   // Stellrückmeldungen
   "UP_CM03.GP03".In.SRM_Saugseite_auf := "E_SRM_CM03.QM33_auf" AND NOT "E_SRM_CM03.QM33_zu";
   "UP_CM03.GP03".In.SRM_Saugseite_zu := "E_SRM_CM03.QM33_zu" AND NOT "E_SRM_CM03.QM33_auf";
   "UP_CM03.GP03".In.SRM_Druckseite_auf := "E_SRM_CM03.QM34_auf" AND NOT "E_SRM_CM03.QM34_zu";
   "UP_CM03.GP03".In.SRM_Druckseite_zu := "E_SRM_CM03.QM34_zu" AND NOT "E_SRM_CM03.QM34_auf";

   "UP_CM03.GP03".In.GW_p_UP := "E_GW_p_CM03.BP05";
   // TW senkt
   "UP_CM03.GP03".In.TW_senkt := ("DB_POS".POS[7].FW_Senkt OR "DB_POS".POS[8].FW_Senkt OR "DB_POS".POS[9].FW_Senkt
   OR "DB_POS".POS[10].FW_Senkt OR "DB_POS".POS[11].FW_Senkt OR "DB_POS".POS[12].FW_Senkt) AND "DI_FW_1".ZST.Mittig;

   // Frequenzumrichter [Index 3]
   "UP_CM03.GP03".In.FU_speed := "FU_In_Out".FU[3].PE.Speed;
   "UP_CM03.GP03".In.FU_betriebsbereit := "FU_In_Out".FU[3].PE.Statusbyte.Bereit;
   "UP_CM03.GP03".In.FU_Stoerung := "FU_In_Out".FU[3].PE.Statusbyte.Stoer;
   "UP_CM03.GP03".Param.SW_Hand := "Panel".UP_CM03.SW_Hand;
   "UP_CM03.GP03".Param.SW_Auto_AZ := "Panel".UP_CM03.SW_Auto_AZ;
   "UP_CM03.GP03".Param.SW_Auto_aAZ := "Panel".UP_CM03.SW_Auto_aAZ;

   // Hand
   "UP_CM03.GP03".In.Ein := "Panel".UP_CM03.Ein;
   // Auto
   "UP_CM03.GP03".In.Auto := FALSE; // "Panel".UP_CM03.Auto;
   // Betriebsart
   "UP_CM03.GP03".In.Betriebsart := "Panel".UP_CM03.BA;
   // Spülzeit
   "UP_CM03.GP03".Param.Spülzeit := DINT_TO_TIME(INT_TO_DINT("Panel".UP_CM03.Sp_Ventil.Sollzeit) * 1000);
   // Drucktest
   "UP_CM03.GP03".Param.DT_Druckaufbau := T#1m;
   "UP_CM03.GP03".Param.SW_Drucktest := "Panel".UP_CM03.Drucktest.Solldruck;
   "UP_CM03.GP03".Param.DT_Testzeit := DINT_TO_TIME(INT_TO_DINT("Panel".UP_CM03.Drucktest.Sollzeit) * 1000);


   // --> Panel
   "Panel".CM03.Niv_TGS := "UP_CM03.GP03".In.Niv_TLS;
   "Panel".CM03.Niv_Min := "UP_CM03.GP03".In.Niv_min;
   "Panel".CM03.GW_p_UP := "UP_CM03.GP03".In.GW_p_UP;
   "Panel".CM03.Niv_Proz := "UP_CM03.GP03".Zst.Niveau;
   "Panel".UP_CM03.Sp_Ventil.Restzeit := TIME_TO_INT("UP_CM03.GP03".Zst.Restzeit_Spülen / 1000);
   "Panel".UP_CM03.Drucktest.Restzeit := TIME_TO_INT("UP_CM03.GP03".Zst.Restzeit_DT / 1000);
   "Panel".UP_CM03.Drucktest.Schritt := "UP_CM03.GP03".Zst.Status_DT;
   "Panel".UP_CM03.Status := "UP_CM03.GP03".Zst.Status_GP0x;
   "Panel".UP_CM03.speed := "UP_CM03.GP03".Zst.speed;
   "Panel".UP_CM03.Bedienung_Erlaubt := "UP_CM03.GP03".Zst.Bedienung_erlaubt;
END_REGION

REGION Network 6 (SCL): CM04
   "UP_CM04.GP06".Param.Name := 'UP_CM04.GP06';
   // Niveaus
   "UP_CM04.GP06".In.Niv_TLS := "E_Niv_TLS_CM04.BL14";
   "UP_CM04.GP06".In.Niv_min := "E_Niv_Min_CM04.BL13";
   "UP_CM04.GP06".In.Frg_Niv_CM05 := NOT "Pu_CM05.GP11_DB".In."Niv_max_CM05.BL01" AND NOT "Pu_CM05.GP11_DB".In."Niv_Uel_CM05.BL05";
   "UP_CM04.GP06".In.ext_Freigabe := "E_Al_Gas_ok" AND NOT "E_Not-Strom";
   // Ist-Druck
   "UP_CM04.GP06".In.Druck_Pumpe := "Panel".IW."p_CM04.BP08";

   // Stellrückmeldungen
   "UP_CM04.GP06".In.SRM_Saugseite_auf := "E_SRM_CM04.QM72_auf" AND NOT "E_SRM_CM04.QM72_zu";
   "UP_CM04.GP06".In.SRM_Saugseite_zu := "E_SRM_CM04.QM72_zu" AND NOT "E_SRM_CM04.QM72_auf";
   "UP_CM04.GP06".In.SRM_Druckseite_auf := "E_SRM_CM04.QM73_auf" AND NOT "E_SRM_CM04.QM73_zu";
   "UP_CM04.GP06".In.SRM_Druckseite_zu := "E_SRM_CM04.QM73_zu" AND NOT "E_SRM_CM04.QM73_auf";

   "UP_CM04.GP06".In.GW_p_UP := "E_GW_p_CM04.BP08";

   // TW senkt
   "UP_CM04.GP06".In.TW_senkt := ("DB_POS".POS[19].FW_Senkt OR "DB_POS".POS[20].FW_Senkt OR "DB_POS".POS[21].FW_Senkt
   OR "DB_POS".POS[22].FW_Senkt OR "DB_POS".POS[23].FW_Senkt OR "DB_POS".POS[24].FW_Senkt) AND "DI_FW_1".ZST.Mittig;

   // Frequenzumrichter [Index 6]
   "UP_CM04.GP06".In.FU_speed := "FU_In_Out".FU[6].PE.Speed;
   "UP_CM04.GP06".In.FU_betriebsbereit := "FU_In_Out".FU[6].PE.Statusbyte.Bereit;
   "UP_CM04.GP06".In.FU_Stoerung := "FU_In_Out".FU[6].PE.Statusbyte.Stoer;
   "UP_CM04.GP06".Param.SW_Hand := "Panel".UP_CM04.SW_Hand;
   "UP_CM04.GP06".Param.SW_Auto_AZ := "Panel".UP_CM04.SW_Auto_AZ;
   "UP_CM04.GP06".Param.SW_Auto_aAZ := "Panel".UP_CM04.SW_Auto_aAZ;

   // Hand
   "UP_CM04.GP06".In.Ein := "Panel".UP_CM04.Ein;
   // Auto
   "UP_CM04.GP06".In.Auto := FALSE; // "Panel".UP_CM04.Auto;
   // Betriebsart
   "UP_CM04.GP06".In.Betriebsart := "Panel".UP_CM04.BA;

   // Spülzeit
   "UP_CM04.GP06".Param.Spülzeit := DINT_TO_TIME(INT_TO_DINT("Panel".UP_CM04.Sp_Ventil.Sollzeit) * 1000);
   // Drucktest
   "UP_CM04.GP06".Param.DT_Druckaufbau := T#1m;
   "UP_CM04.GP06".Param.SW_Drucktest := "Panel".UP_CM04.Drucktest.Solldruck;
   "UP_CM04.GP06".Param.DT_Testzeit := DINT_TO_TIME(INT_TO_DINT("Panel".UP_CM04.Drucktest.Sollzeit) * 1000);

   // --> Panel
   "Panel".CM04.Niv_TGS := "UP_CM04.GP06".In.Niv_TLS;
   "Panel".CM04.Niv_Min := "UP_CM04.GP06".In.Niv_min;
   "Panel".CM04.GW_p_UP := "UP_CM04.GP06".In.GW_p_UP;
   "Panel".CM04.Niv_Proz := "UP_CM04.GP06".Zst.Niveau;
   "Panel".UP_CM04.Sp_Ventil.Restzeit := TIME_TO_INT("UP_CM04.GP06".Zst.Restzeit_Spülen / 1000);
   "Panel".UP_CM04.Drucktest.Restzeit := TIME_TO_INT("UP_CM04.GP06".Zst.Restzeit_DT / 1000);
   "Panel".UP_CM04.Drucktest.Schritt := "UP_CM04.GP06".Zst.Status_DT;
   "Panel".UP_CM04.Status := "UP_CM04.GP06".Zst.Status_GP0x;
   "Panel".UP_CM04.speed := "UP_CM04.GP06".Zst.speed;
   "Panel".UP_CM04.Bedienung_Erlaubt := "UP_CM04.GP06".Zst.Bedienung_erlaubt;
END_REGION

REGION Network 7 (SCL): CM05
   // Motorschutzschalter
   "Pu_CM05.GP11_DB".In.MSS_ok := "E_MSS_ok_CM05.GP11";
   // Druckschalter
   "Pu_CM05.GP11_DB".In.GW_p := "E_GW_p_CM05.BP09";
   // Ist-Druck
   "Pu_CM05.GP11_DB".In.Druck_Pumpe :="Panel".IW."p_CM05.BP09";

   // Niveaus
   "Pu_CM05.GP11_DB".In."Niv_max_CM05.BL01" := "E_Niv_max_CM05.BL01";
   "Pu_CM05.GP11_DB".In."Niv_min_CM05.BL02" := "E_Niv_min_CM05.BL02";
   "Pu_CM05.GP11_DB".In."Niv_TLS_CM05.BL03" := "E_Niv_TLS_CM05.BL03";
   "Pu_CM05.GP11_DB".In."Niv_Uel_CM05.BL05" :=  NOT "E_Niv_Uel_CM05.BL12";

   // Stellrückmeldungen
   "Pu_CM05.GP11_DB".In."SRM_CM05.QM61_auf" := "E_SRM_CM05.QM61_auf" AND NOT "E_SRM_CM05.QM61_zu";
   "Pu_CM05.GP11_DB".In."SRM_CM05.QM61_zu" := "E_SRM_CM05.QM61_zu" AND NOT "E_SRM_CM05.QM61_auf";
   "Pu_CM05.GP11_DB".In."SRM_CM05.QM64_auf" := "E_SRM_CM05.QM64_auf" AND NOT "E_SRM_CM05.QM64_zu";
   "Pu_CM05.GP11_DB".In."SRM_CM05.QM64_zu" := "E_SRM_CM05.QM64_zu"  AND NOT "E_SRM_CM05.QM64_auf";

   // Neutra
   "Pu_CM05.GP11_DB".In.AWA_ok := "E_AWA_ok";
   "Pu_CM05.GP11_DB".In.Frg_AWA := "E_Frg_AWA";
   // Hand
   "Pu_CM05.GP11_DB".In.Ein := "Panel".Pu_CM05.Ein;
   // Auto
   "Pu_CM05.GP11_DB".In.Auto := "Panel".Pu_CM05.Auto;
   // Betriebsart
   "Pu_CM05.GP11_DB".In.Betriebsart := "Panel".Pu_CM05.BA;
   // Spülzeit
   "Pu_CM05.GP11_DB".Param.Spülzeit := DINT_TO_TIME(INT_TO_DINT("Panel".Pu_CM05.Sp_Ventil.Sollzeit) * 1000);
   // Drucktest
   "Pu_CM05.GP11_DB".Param.DT_Druckaufbau := T#1m;
   "Pu_CM05.GP11_DB".Param.SW_Drucktest := "Panel".Pu_CM05.Drucktest.Solldruck;
   "Pu_CM05.GP11_DB".Param.DT_Testzeit := DINT_TO_TIME(INT_TO_DINT("Panel".Pu_CM05.Drucktest.Sollzeit) * 1000);

   // --> Panel
   "Panel".CM05.GW_p_Pu := "Pu_CM05.GP11_DB".In.GW_p;
   "Panel".CM05.Niv_Proz := "Pu_CM05.GP11_DB".Zst.Niveau;
   "Panel".CM05.Niv_TGS := "Pu_CM05.GP11_DB".In."Niv_TLS_CM05.BL03";
   "Panel".CM05.Niv_Min := "Pu_CM05.GP11_DB".In."Niv_min_CM05.BL02";
   "Panel".CM05.Niv_max := "Pu_CM05.GP11_DB".In."Niv_max_CM05.BL01";
   "Panel".CM05.Niv_Uel := "Pu_CM05.GP11_DB".In."Niv_Uel_CM05.BL05";
   "Panel".Pu_CM05.Sp_Ventil.Restzeit := TIME_TO_INT("Pu_CM05.GP11_DB".Zst.Restzeit_Spülen / 1000);
   "Panel".Pu_CM05.Drucktest.Restzeit := TIME_TO_INT("Pu_CM05.GP11_DB".Zst.Restzeit_DT / 1000);
   "Panel".Pu_CM05.Drucktest.Schritt := "Pu_CM05.GP11_DB".Zst.Status_DT;
   "Panel".Pu_CM05.Status := "Pu_CM05.GP11_DB".Zst.Status_GP11;
   "Panel".CM05.AWA_Bereit := "Pu_CM05.GP11_DB".In.AWA_ok;
   "Panel".CM05.Frg_Abpumpen := "Pu_CM05.GP11_DB".In.Frg_AWA;
   "Panel".Pu_CM05.Bedienung_Erlaubt := "Pu_CM05.GP11_DB".Zst.Bedienung_erlaubt;
END_REGION

REGION Network 8 (SCL): CL0x
   //CL01
   // Niveaus
   "Pu_CL01.GP08".In.Frg_Niv_CM05 :=  NOT "Pu_CM05.GP11_DB".In."Niv_max_CM05.BL01" AND NOT "Pu_CM05.GP11_DB".In."Niv_Uel_CM05.BL05";
   "Pu_CL01.GP08".In.Leckage_ok := "E_LS_CL01.BL28";
   // Hand
   "Pu_CL01.GP08".In.Ein :="Panel".Pu_CL01.Ein;
   // Auto
   "Pu_CL01.GP08".In.Auto := "Panel".Pu_CL01.Auto;
   // Betriebsart
   "Pu_CL01.GP08".In.Betriebsart := "Panel".Pu_CL01.BA;
   // Spülzeit
   "Pu_CL01.GP08".Param.Spülzeit := DINT_TO_TIME(INT_TO_DINT("Panel".Pu_CL01.Sp_Ventil.Sollzeit) * 1000);

   // --> Panel
   "Panel".CL0x."LS_CL01.BL28" := NOT "Pu_CL01.GP08".In.Leckage_ok;
   "Panel".CL0x.Niv_Proz_CL01 := "Pu_CL01.GP08".Zst.Niveau;
   "Panel".Pu_CL01.Sp_Ventil.Restzeit := TIME_TO_INT("Pu_CL01.GP08".Zst.Restzeit_Spülen / 1000);
   "Panel".Pu_CL01.Status := "Pu_CL01.GP08".Zst.Status_GP0x;
   "Panel".Pu_CL01.Bedienung_Erlaubt := "Pu_CL01.GP08".Zst.Bedienung_Erlaubt;

   //CL02
   // Niveaus
   "Pu_CL02.GP09".In.Frg_Niv_CM05 :=  NOT "Pu_CM05.GP11_DB".In."Niv_max_CM05.BL01" AND NOT "Pu_CM05.GP11_DB".In."Niv_Uel_CM05.BL05";
   "Pu_CL02.GP09".In.Leckage_ok := "E_LS_CL02.BL29";
   // Hand
   "Pu_CL02.GP09".In.Ein := "Panel".Pu_CL02.Ein;
   // Auto
   "Pu_CL02.GP09".In.Auto := "Panel".Pu_CL02.Auto;
   // Betriebsart
   "Pu_CL02.GP09".In.Betriebsart := "Panel".Pu_CL02.BA;
   // Spülzeit
   "Pu_CL02.GP09".Param.Spülzeit := DINT_TO_TIME(INT_TO_DINT("Panel".Pu_CL02.Sp_Ventil.Sollzeit) * 1000);

   // --> Panel
   "Panel".CL0x."LS_CL02.BL29" := NOT  "Pu_CL02.GP09".In.Leckage_ok;
   "Panel".CL0x.Niv_Proz_CL02 := "Pu_CL02.GP09".Zst.Niveau;
   "Panel".Pu_CL02.Sp_Ventil.Restzeit := TIME_TO_INT("Pu_CL02.GP09".Zst.Restzeit_Spülen / 1000);
   "Panel".Pu_CL02.Status := "Pu_CL02.GP09".Zst.Status_GP0x;
   "Panel".Pu_CL02.Bedienung_Erlaubt := "Pu_CL02.GP09".Zst.Bedienung_Erlaubt;
END_REGION

REGION Network 9 (SCL): GP01
   // Versorgung
   //Niveaus
   "Pu_GP01.GP13".In.Niv_min := "E_Niv_min_GP01.BL17";
   "Pu_GP01.GP13".In.Niv_max := NOT "E_Niv_max_GP01.BL20";
   "Pu_GP01.GP13".In.Niveau := INT_TO_USINT(REAL_TO_INT("Panel".IW."Niv_GP01.BL30"));
   // Leckagesensoren
   "Pu_GP01.GP13".In.Leckage_Pumpe_ok := NOT "E_LS_GP01.BL15";
   "Pu_GP01.GP13".In.Leckage_PFA_Uebergang_ok := "E_LS_GP01.BL16";
   "Pu_GP01.GP13".In.Leckage_Doppelrohr_ok := "E_LS_GP01.BL19";
   "Pu_GP01.GP13".In.Leckage_Uml_Tunnel_ok := "E_LS_GP01.BL34";
   "Pu_GP01.GP13".In.Leckage_Doppelschlauch_ok := TRUE; // nur GP02
   "Pu_GP01.GP13".In.kein_Gas_Alarm := "E_Al_Gas_ok";

   "Pu_GP01.GP13".In.Niv_Min_CM01 := "E_Niv_Min_CM01.BL03";
   "Pu_GP01.GP13".In.Niv_Max_CM01 := "E_Niv_Max_CM01.BL02";
   "Pu_GP01.GP13".In.Niv_Übervoll_CM01 := NOT "E_Niv_UeL_CM01.BL01";
   "Pu_GP01.GP13".In.Niv_Min_CM02 := "E_Niv_Min_CM02.BL10";
   "Pu_GP01.GP13".In.Niv_Max_CM02 := "E_Niv_Max_CM02.BL09";
   "Pu_GP01.GP13".In.Niv_Übervoll_CM02 := NOT "E_Niv_UeL_CM02.BL08";
   "Pu_GP01.GP13".In.Frg_Niv_CM05 := NOT "Pu_CM05.GP11_DB".In."Niv_max_CM05.BL01" AND NOT "Pu_CM05.GP11_DB".In."Niv_Uel_CM05.BL05";

   // Stellrückmeldungen
   "Pu_GP01.GP13".In.SRM_Saugseite_auf := "E_SRM_GP01.QM15_auf" AND NOT "E_SRM_GP01.QM15_zu";
   "Pu_GP01.GP13".In.SRM_Saugseite_zu := "E_SRM_GP01.QM15_zu" AND NOT "E_SRM_GP01.QM15_auf";
   "Pu_GP01.GP13".In.SRM_Druckseite_auf := "E_SRM_GP01.QM18_auf" AND NOT "E_SRM_GP01.QM18_zu";
   "Pu_GP01.GP13".In.SRM_Druckseite_zu := "E_SRM_GP01.QM18_zu" AND NOT "E_SRM_GP01.QM18_auf";
   "Pu_GP01.GP13".In.SRM_Eingang_Spülltg_auf := "E_SRM_GP01.QM16_auf" AND NOT "E_SRM_GP01.QM16_zu";
   "Pu_GP01.GP13".In.SRM_Eingang_Spülltg_zu := "E_SRM_GP01.QM16_zu" AND NOT "E_SRM_GP01.QM16_auf";
   "Pu_GP01.GP13".In.SRM_Ausgang_Spülltg_auf := "E_SRM_GP01.QM17_auf" AND NOT "E_SRM_GP01.QM17_zu";
   "Pu_GP01.GP13".In.SRM_Ausgang_Spülltg_zu := "E_SRM_GP01.QM17_zu" AND NOT "E_SRM_GP01.QM17_auf";
   "Pu_GP01.GP13".In.SRM_Versogung_UV01_auf := "E_SRM_GP01.QM22_auf" AND NOT "E_SRM_GP01.QM22_zu";
   "Pu_GP01.GP13".In.SRM_Versogung_UV01_zu := "E_SRM_GP01.QM22_zu" AND NOT "E_SRM_GP01.QM22_auf";
   "Pu_GP01.GP13".In.SRM_UV01_CM01_auf := "E_SRM_GP01.QM20_auf" AND NOT "E_SRM_GP01.QM20_zu";
   "Pu_GP01.GP13".In.SRM_UV01_CM01_zu := "E_SRM_GP01.QM20_zu" AND NOT "E_SRM_GP01.QM20_auf";
   "Pu_GP01.GP13".In.SRM_UV01_CM02_auf := "E_SRM_GP01.QM19_auf" AND NOT "E_SRM_GP01.QM19_zu";
   "Pu_GP01.GP13".In.SRM_UV01_CM02_zu := "E_SRM_GP01.QM19_zu" AND NOT "E_SRM_GP01.QM19_auf";

   "Pu_GP01.GP13".In.IBC_vorhanden := "E_S_IBC_GP01.BG21";
   "Pu_GP01.GP13".In.Tuer_vorn_zu := "DB_PNOZ_IN_Out".In.Tuer_zu_vorn_GP01;
   "Pu_GP01.GP13".In.Tuer_seitlich_zu := "DB_PNOZ_IN_Out".In.Tuer_zu_Seite_GP01;

   "Pu_GP01.GP13".In.GW_Dfl := "E_GW_Dfl_GP01.BF01";
   "Pu_GP01.GP13".In.Imp_Dfl := "E_Imp_GP01.BF01";
   "Pu_GP01.GP13".In.Quitt_Al_Dfl := "DB_ANLAGE".IN.Quitt_Err;
   "Pu_GP01.GP13".In.Dfl := "Panel".IW."Dfl_GP01.BF01";

   // Hand
   "Pu_GP01.GP13".In.Ein := "Panel".Pu_Vers_GP01.Ein;
   // Auto
   "Pu_GP01.GP13".In.Auto := "Panel".Pu_Vers_GP01.Auto;
   // Betriebsart
   "Pu_GP01.GP13".In.Betriebsart := "Panel".Pu_Vers_GP01.BA;
   // Spülzeit
   "Pu_GP01.GP13".Param.Spülzeit := DINT_TO_TIME(INT_TO_DINT("Panel".Pu_Vers_GP01.Sp_Ventil.Sollzeit) * 1000);

   // --> Panel
   "Panel".GP01.Niv_leer := "Pu_GP01.GP13".In.Niv_min;
   "Panel".GP01.Niv_max := "Pu_GP01.GP13".In.Niv_max;
   "Panel".GP01.IBC_vorhanden := "Pu_GP01.GP13".In.IBC_vorhanden;
   "Panel".GP01.Tür_zu_vorn := "Pu_GP01.GP13".In.Tuer_vorn_zu;
   "Panel".GP01.Tür_zu_seitlich := "Pu_GP01.GP13".In.Tuer_seitlich_zu;

   "Panel".GP01.LS_Pumpe := NOT "Pu_GP01.GP13".In.Leckage_Pumpe_ok;
   "Panel".GP01.LS_Doppelrohr_BL19 := NOT "Pu_GP01.GP13".In.Leckage_Doppelrohr_ok;
   "Panel".GP01.LS_PFA_Übergang := NOT "Pu_GP01.GP13".In.Leckage_PFA_Uebergang_ok;
   "Panel".GP01.LS_Uml_Tunnel := NOT "Pu_GP01.GP13".In.Leckage_Uml_Tunnel_ok;

   "Panel".GP01.Niv_Proz := "Pu_GP01.GP13".In.Niveau;

   "Panel".GP01.Versorgung := "Pu_GP01.GP13".In.Betriebsart < 4;
   "Panel".GP01.Entsorgung := "Pu_GP01.GP13".In.Betriebsart = 4;


   "Panel".Pu_Vers_GP01.Status := "Pu_GP01.GP13".Zst.Status_GP0x;
   "Panel".Pu_Vers_GP01.Sp_Ventil.Restzeit := TIME_TO_INT("Pu_GP01.GP13".Zst.Restzeit_Spülen / 1000);
   "Panel".Pu_Vers_GP01.Bedienung_Erlaubt := "Pu_GP01.GP13".Zst.Bedienung_erlaubt;
   //-----------------------------------------------------------------------------------------------------------------------------------------
   // Abpumpen
   // Niveaus
   "Pu_GP01.GP12".In.Frg_Niv_CM05 :=  NOT "Pu_CM05.GP11_DB".In."Niv_max_CM05.BL01" AND NOT "Pu_CM05.GP11_DB".In."Niv_Uel_CM05.BL05";
   "Pu_GP01.GP12".In.Leckage_ok := "E_LS_GP01.BL18";
   // Hand
   "Pu_GP01.GP12".In.Ein := "Panel".Pu_Entl_GP01.Ein;
   // Auto
   "Pu_GP01.GP12".In.Auto := "Panel".Pu_Entl_GP01.Auto;
   // Betriebsart
   "Pu_GP01.GP12".In.Betriebsart := "Panel".Pu_Entl_GP01.BA;
   // Spülzeit
   "Pu_GP01.GP12".Param.Spülzeit := DINT_TO_TIME(INT_TO_DINT("Panel".Pu_Entl_GP01.Sp_Ventil.Sollzeit) * 1000);

   // --> Panel
   "Panel".GP01.LS_PuSu := NOT "Pu_GP01.GP12".In.Leckage_ok;
   "Panel".Pu_Entl_GP01.Sp_Ventil.Restzeit := TIME_TO_INT("Pu_GP01.GP12".Zst.Restzeit_Spülen / 1000);
   "Panel".Pu_Entl_GP01.Status := "Pu_GP01.GP12".Zst.Status_GP0x;
   "Panel".Pu_Entl_GP01.Bedienung_Erlaubt := "Pu_GP01.GP12".Zst.Bedienung_Erlaubt;
END_REGION

REGION Network 10 (SCL): GP02
   // Versorgung
   //Niveaus
   "Pu_GP02.GP10".In.Niv_min := "E_Niv_min_GP02.BL24";
   "Pu_GP02.GP10".In.Niv_max := NOT "E_Niv_max_GP02.BL23";
   "Pu_GP02.GP10".In.Niveau := INT_TO_USINT(REAL_TO_INT("Panel".IW."Niv_GP02.BL31"));
   // Leckagesensoren
   "Pu_GP02.GP10".In.Leckage_Pumpe_ok := NOT "E_LS_GP02.BL27";
   "Pu_GP02.GP10".In.Leckage_PFA_Uebergang_ok := "E_LS_GP02.BL25";
   "Pu_GP02.GP10".In.Leckage_Doppelrohr_ok := "E_LS_GP01.BL19";
   "Pu_GP02.GP10".In.Leckage_Uml_Tunnel_ok := TRUE; // nur GP01
   "Pu_GP02.GP10".In.Leckage_Doppelschlauch_ok := "E_LS_GP02.BL32";
   "Pu_GP02.GP10".In.kein_Gas_Alarm := "E_Al_Gas_ok";

   "Pu_GP02.GP10".In.Niv_Min_CM01 := "E_Niv_Min_CM01.BL03";
   "Pu_GP02.GP10".In.Niv_Max_CM01 := "E_Niv_Max_CM01.BL02";
   "Pu_GP02.GP10".In.Niv_Übervoll_CM01 := NOT "E_Niv_UeL_CM01.BL01";
   "Pu_GP02.GP10".In.Niv_Min_CM02 := "E_Niv_Min_CM02.BL10";
   "Pu_GP02.GP10".In.Niv_Max_CM02 := "E_Niv_Max_CM02.BL09";
   "Pu_GP02.GP10".In.Niv_Übervoll_CM02 := NOT "E_Niv_UeL_CM02.BL08";
   "Pu_GP02.GP10".In.Frg_Niv_CM05 := NOT "Pu_CM05.GP11_DB".In."Niv_max_CM05.BL01" AND NOT "Pu_CM05.GP11_DB".In."Niv_Uel_CM05.BL05";

   // Stellrückmeldungen
   "Pu_GP02.GP10".In.SRM_Saugseite_auf := "E_SRM_GP02.QM38_auf" AND NOT "E_SRM_GP02.QM38_zu";
   "Pu_GP02.GP10".In.SRM_Saugseite_zu := "E_SRM_GP02.QM38_zu" AND NOT "E_SRM_GP02.QM38_auf";
   "Pu_GP02.GP10".In.SRM_Druckseite_auf := "E_SRM_GP02.QM40_auf" AND NOT "E_SRM_GP02.QM40_zu";
   "Pu_GP02.GP10".In.SRM_Druckseite_zu := "E_SRM_GP02.QM40_zu" AND NOT "E_SRM_GP02.QM40_auf";
   "Pu_GP02.GP10".In.SRM_Eingang_Spülltg_auf := "E_SRM_GP02.QM39_auf" AND NOT "E_SRM_GP02.QM39_zu";
   "Pu_GP02.GP10".In.SRM_Eingang_Spülltg_zu := "E_SRM_GP02.QM39_zu" AND NOT "E_SRM_GP02.QM39_auf";
   "Pu_GP02.GP10".In.SRM_Ausgang_Spülltg_auf := "E_SRM_GP02.QM42_auf" AND NOT "E_SRM_GP02.QM42_zu";
   "Pu_GP02.GP10".In.SRM_Ausgang_Spülltg_zu := "E_SRM_GP02.QM42_zu" AND NOT "E_SRM_GP02.QM42_auf";
   "Pu_GP02.GP10".In.SRM_Versogung_UV01_auf := "E_SRM_GP01.QM21_auf" AND NOT "E_SRM_GP01.QM21_zu";
   "Pu_GP02.GP10".In.SRM_Versogung_UV01_zu := "E_SRM_GP01.QM21_zu" AND NOT "E_SRM_GP01.QM21_auf";
   "Pu_GP02.GP10".In.SRM_UV01_CM01_auf := "E_SRM_GP01.QM20_auf" AND NOT "E_SRM_GP01.QM20_zu";
   "Pu_GP02.GP10".In.SRM_UV01_CM01_zu := "E_SRM_GP01.QM20_zu" AND NOT "E_SRM_GP01.QM20_auf";
   "Pu_GP02.GP10".In.SRM_UV01_CM02_auf := "E_SRM_GP01.QM19_auf" AND NOT "E_SRM_GP01.QM19_zu";
   "Pu_GP02.GP10".In.SRM_UV01_CM02_zu := "E_SRM_GP01.QM19_zu" AND NOT "E_SRM_GP01.QM19_auf";

   "Pu_GP02.GP10".In.IBC_vorhanden := "E_S_IBC_GP02.BG22";
   "Pu_GP02.GP10".In.Tuer_vorn_zu := "DB_PNOZ_IN_Out".In.Tuer_zu_vorn_GP02;
   "Pu_GP02.GP10".In.Tuer_seitlich_zu := TRUE;

   "Pu_GP02.GP10".In.GW_Dfl := "E_GW_Dfl_GP01.BF01";
   "Pu_GP02.GP10".In.Imp_Dfl := "E_Imp_GP01.BF01";
   "Pu_GP02.GP10".In.Quitt_Al_Dfl := "DB_ANLAGE".IN.Quitt_Err;
   "Pu_GP02.GP10".In.Dfl := "Panel".IW."Dfl_GP01.BF01";
   "Pu_GP02.GP10".In.Niveau := INT_TO_USINT(REAL_TO_INT("Panel".IW."Niv_GP02.BL31"));

   // Hand
   "Pu_GP02.GP10".In.Ein := "Panel".Pu_Vers_GP02.Ein;
   // Auto
   "Pu_GP02.GP10".In.Auto := "Panel".Pu_Vers_GP02.Auto;
   // Betriebsart
   "Pu_GP02.GP10".In.Betriebsart := "Panel".Pu_Vers_GP02.BA;
   // Spülzeit
   "Pu_GP02.GP10".Param.Spülzeit := DINT_TO_TIME(INT_TO_DINT("Panel".Pu_Vers_GP02.Sp_Ventil.Sollzeit) * 1000);

   // --> Panel
   "Panel".GP02.Niv_leer := "Pu_GP02.GP10".In.Niv_min;
   "Panel".GP02.Niv_max := "Pu_GP02.GP10".In.Niv_max;
   "Panel".GP02.IBC_vorhanden := "Pu_GP02.GP10".In.IBC_vorhanden;

   "Panel".GP02.Tür_zu_seitlich := "Pu_GP02.GP10".In.Tuer_seitlich_zu;

   "Panel".GP02.LS_Doppelschlauch_BL32 := NOT "E_LS_GP02.BL32";
   "Panel".GP02.LS_Doppelschlauch_BL33 := NOT "E_LS_GP02.BL33";
   "Panel".GP02.LS_Doppelrohr_BL26 := NOT "E_LS_GP02.BL26";
   "Panel".GP02.LS_Pumpe := NOT "Pu_GP02.GP10".In.Leckage_Pumpe_ok;
   "Panel".GP02.LS_PFA_Übergang := NOT "Pu_GP02.GP10".In.Leckage_PFA_Uebergang_ok;
   "Panel".GP02.Niv_Proz := "Pu_GP02.GP10".In.Niveau;

   "Panel".GP02.Versorgung := "Pu_GP02.GP10".In.Betriebsart < 4;
   "Panel".GP02.Entsorgung := "Pu_GP02.GP10".In.Betriebsart = 4;

   "Panel".Pu_Vers_GP02.Status := "Pu_GP02.GP10".Zst.Status_GP0x;
   "Panel".Pu_Vers_GP02.Sp_Ventil.Restzeit := TIME_TO_INT("Pu_GP02.GP10".Zst.Restzeit_Spülen / 1000);
   "Panel".Pu_Vers_GP02.Bedienung_Erlaubt := "Pu_GP02.GP10".Zst.Bedienung_erlaubt;
   //-----------------------------------------------------------------------------------------------------------------------------------------

   // Abpumpen
   // Niveaus
   "Pu_GP02.GP07".In.Frg_Niv_CM05 :=  NOT "Pu_CM05.GP11_DB".In."Niv_max_CM05.BL01" AND NOT "Pu_CM05.GP11_DB".In."Niv_Uel_CM05.BL05";
   "Pu_GP02.GP07".In.Leckage_ok := "E_LS_GP02.BL21";
   // Hand
   "Pu_GP02.GP07".In.Ein := "Panel".Pu_Entl_GP02.Ein;
   // Auto
   "Pu_GP02.GP07".In.Auto := "Panel".Pu_Entl_GP02.Auto;
   // Betriebsart
   "Pu_GP02.GP07".In.Betriebsart := "Panel".Pu_Entl_GP02.BA;
   // Spülzeit
   "Pu_GP02.GP07".Param.Spülzeit := DINT_TO_TIME(INT_TO_DINT("Panel".Pu_Entl_GP02.Sp_Ventil.Sollzeit) * 1000);

   // --> Panel
   "Panel".GP02.LS_PuSu := NOT "Pu_GP02.GP07".In.Leckage_ok;
   "Panel".Pu_Entl_GP02.Sp_Ventil.Restzeit := TIME_TO_INT("Pu_GP02.GP07".Zst.Restzeit_Spülen / 1000);
   "Panel".Pu_Entl_GP02.Status := "Pu_GP02.GP07".Zst.Status_GP0x;
   "Panel".Pu_Entl_GP02.Bedienung_Erlaubt := "Pu_GP02.GP07".Zst.Bedienung_Erlaubt;
END_REGION
END_FUNCTION

FUNCTION "FC_SIMULATION" : Void   // FC200, STL
TITLE = SIMULATION
{ S7_Optimized_Access := 'FALSE' }
AUTHOR : RE
// stored: AutoNumber false
   VAR_TEMP
      count : Int;
      AnzahlWT : Int;
      Faktor : Real;
      TR3 : Real;
      ErrInf : Byte;
      ON : Bool;
      OFF : Bool;
      dummy : Bool;
      Takt : Bool;
      BE_Auto : Bool;
      low : Bool;
      "return" : Bool;
      S01 : Bool;
      S02 : Bool;
      S03 : Bool;
      S04 : Bool;
      S05 : Bool;
      S06 : Bool;
      S07 : Bool;
      S00 : Bool;
      HZ1 : Bool;   // Heizung 1 an
      HZ2 : Bool;   // Heizung 2 an
      KHL : Bool;   // Kühlung an
      TypExo : Bool;   // Bad mit Kühlregler
      v0 : Bool;
   END_VAR
BEGIN

NETWORK
TITLE = Simulation Anlage

      AN    "DB_ANLAGE".BA.Simulation;
      BEC;

//-------------------------
//Beladestände simulieren
//-------------------------
      L     "DB_POS".POS[25].WT_DB;
      L     0;
      <>I;
      S     "DB_BE_Stand".Stand[1].IN_Belegt;

      A     "DB_POS".POS[25].FW_Hebt;
      AN    "DI_FW_1".ZST.low_SU_li;
      R     "DB_BE_Stand".Stand[1].IN_Belegt;

      SET;
      =     "DB_BE_Stand".Stand[1].IN_innen;
      =     "DB_BE_Stand".Stand[1].IN_aussen;
      =     "DB_BE_Stand".Stand[1].verriegelt;
      =     "DB_BE_Stand".Stand[1].IN_Freigabe;

      L     "DB_POS".POS[26].WT_DB;
      L     0;
      <>I;
      S     "DB_BE_Stand".Stand[2].IN_Belegt;

      A     "DB_POS".POS[26].FW_Hebt;
      AN    "DI_FW_1".ZST.low_SU_re;
      R     "DB_BE_Stand".Stand[2].IN_Belegt;

      SET;
      =     "DB_BE_Stand".Stand[2].IN_innen;
      =     "DB_BE_Stand".Stand[2].IN_aussen;
      =     "DB_BE_Stand".Stand[2].verriegelt;
      =     "DB_BE_Stand".Stand[2].IN_Freigabe;

      L     "DB_POS".POS[27].WT_DB;
      L     0;
      <>I;
      S     "DB_BE_Stand".Stand[3].IN_Belegt;

      A     "DB_POS".POS[27].FW_Hebt;
      AN    "DI_FW_1".ZST.low_SU_li;
      R     "DB_BE_Stand".Stand[3].IN_Belegt;

      SET;
      =     "DB_BE_Stand".Stand[3].IN_innen;
      =     "DB_BE_Stand".Stand[3].IN_aussen;
      =     "DB_BE_Stand".Stand[3].verriegelt;
      =     "DB_BE_Stand".Stand[3].IN_Freigabe;

      L     "DB_POS".POS[28].WT_DB;
      L     0;
      <>I;
      S     "DB_BE_Stand".Stand[2].IN_Belegt;

      A     "DB_POS".POS[28].FW_Hebt;
      AN    "DI_FW_1".ZST.low_SU_re;
      R     "DB_BE_Stand".Stand[4].IN_Belegt;

      SET;
      =     "DB_BE_Stand".Stand[4].IN_innen;
      =     "DB_BE_Stand".Stand[4].IN_aussen;
      =     "DB_BE_Stand".Stand[4].verriegelt;
      =     "DB_BE_Stand".Stand[4].IN_Freigabe;

      L     "DB_POS".POS[29].WT_DB;
      L     0;
      <>I;
      S     "DB_BE_Stand".Stand[5].IN_Belegt;

      A     "DB_POS".POS[29].FW_Hebt;
      AN    "DI_FW_1".ZST.low_SU_li;
      R     "DB_BE_Stand".Stand[5].IN_Belegt;

      SET;
      =     "DB_BE_Stand".Stand[5].IN_innen;
      =     "DB_BE_Stand".Stand[5].IN_aussen;
      =     "DB_BE_Stand".Stand[5].verriegelt;
      =     "DB_BE_Stand".Stand[5].IN_Freigabe;

      L     "DB_POS".POS[30].WT_DB;
      L     0;
      <>I;
      S     "DB_BE_Stand".Stand[6].IN_Belegt;

      A     "DB_POS".POS[30].FW_Hebt;
      AN    "DI_FW_1".ZST.low_SU_re;
      R     "DB_BE_Stand".Stand[6].IN_Belegt;

      SET;
      =     "DB_BE_Stand".Stand[6].IN_innen;
      =     "DB_BE_Stand".Stand[6].IN_aussen;
      =     "DB_BE_Stand".Stand[6].verriegelt;
      =     "DB_BE_Stand".Stand[6].IN_Freigabe;



NETWORK
TITLE = Transportsystem
//****************************************
//           Transportsystem
//****************************************
      L     S5T#2S;
      A     "DB_ANLAGE".IN.S_Not_Aus;
      SF    "T_Verz_NotAus";

      SET;
      =     "DI_FW_1".IN.Laser_on;

//------------------------------------
//             Fahrwagen 1
//------------------------------------
      SET;
      =     "DI_FW_1".IN.Laser_on;

//Stellung Unten
      L     "DI_FW_1".ZST.HubInc_li;
      L     "DI_FW_1".PAR.Hub.Ebene0;
      -D;
      DTR;
      ABS;
      RND;
      L     "DI_FW_1".PAR.Hub.Bereich_Pos;
      <=D;
      =     "DI_FW_1".IN.Unten_li;

//Stellung oben
      L     "DI_FW_1".ZST.HubInc_li;
      L     "DI_FW_1".PAR.Hub.Ebene3;
      -D;
      DTR;
      ABS;
      RND;
      L     "DI_FW_1".PAR.Hub.Bereich_Pos;
      <=D;
      =     "DI_FW_1".IN.Oben_li;

//Stellung Unten
      L     "DI_FW_1".HELP.HubInc_re;
      L     "DI_FW_1".PAR.Hub.Ebene0;
      -D;
      DTR;
      ABS;
      RND;
      L     "DI_FW_1".PAR.Hub.Bereich_Pos;
      <=D;
      =     "DI_FW_1".IN.Unten_re;

//Stellung oben
      L     "DI_FW_1".HELP.HubInc_re;
      L     "DI_FW_1".PAR.Hub.Ebene3;
      -D;
      DTR;
      ABS;
      RND;
      L     "DI_FW_1".PAR.Hub.Bereich_Pos;
      <=D;
      =     "DI_FW_1".IN.Oben_re;

END_FUNCTION

FUNCTION "Analogeingabe" : Void
{ S7_Optimized_Access := 'TRUE' }
VERSION : 0.1
   VAR_TEMP 
      temp_S5Time : S5Time;
      "b-T_Uevoll_VB" : Bool;
      "MW _p_nach Filter_HQ01" : Real;
      "MW _p_nach Filter_HQ02" : Real;
   END_VAR


BEGIN
	// im Sekundentakt
	IF "Imp_1Hz" THEN
	    REGION Leitfähigkeitsmessung
	        // Leitfähigkeit Bypass Filterpumpe
	        "Analogwert"(Deaktiviert:=FALSE,
	                                                                                                                                                                                                                                                                                                                                                                                                                                                                                                                                                                                                                                                                                                                                                                                                                                                                                                                                                                                                                                                                                                                                                                                                                                                                                                                                                                                                                                                                                                                                                                                                                                                                                                                                                                                                                                                                                                                                                                                                                                                                                                                                                                                                                                                                                                                                                                                                                                                                                                                                                                                                                                                                                                                                                                                                                                                                                                                                                                                                                                                                                                                                                                                                                                                                                                                                                                                                                                                                                                                                                                                                                                                                                                                                                                                                                                                                                                                                                                                                                                                                                                                                                                                                                                                                                                                                                                                                                                                                                                                                                                                                                                                                                                                                                                                                                                                                                                                                                                                                                                                                                                                                                                                                                                                                                                                                                                                                                                                                                                                                                                                                                                                                                                                                                                                                                                                                                                                                                                                                                                                                                                                                                                                                                                                                                                                                                                                                                                                                                                                                                                                                                                                                                                                                                                                                                                                                                                                                                                                                                                                                                                                                                                                                                                                                                                                                                                                                                                                                                                                                                                                                                                                                                                                                                                                                                                                                                                                                                                                                                                                                                                                                                                                                                                                                                                                                                                                                                                                                                                                                                                                                                                                                                                                                                                                                                                                                                                                                                                                                                                                                                                                                                                                                                                                                                                                                                                                                                                                                                                                                                                                                                                                                                                                                                                                                                                                                                                                                                                                                                                                                                                                                                                                                                                                                                                                                                                                                                                                                                                                                                                                                                                                                                                                                                                                                                                                                                                                                                                                                                                                                                                                                                                                                                                                                                                                                                                                                                                                                                                                                                                                                                                                                                                                                                                                                                                                                                                                                                                                                                                                                                                                                                                                                                                                                                                                                                                                                                                                                                                                                                                                                                                                                                                                                                                                                                                                                                                                                                                                                                                                                                                                                                                                                                                                                                                                                                                                                                                                                                                                                                                                                                                                                                                                                                                                                                                                                                                                                                                                                                                                                                                                                                                                                                                                                                                                                                                                                                                                                                                                                                                                                                                                                                                                                                                                                                                                                                                                                                                                                                                                                                                                                                                                                                                                                                                                                                                                                                                                                                                                                                                                                                                                                                                                                                                                                                                                                                                                                                                                                                                                                                                                                                                                                                                                                                                                                                                                                                                                                                                                                                                                                                                                                                                                                                                                                                                                                                                                                                                                                                                                                                                                                                                                                                                                                                                                                                                                                                                                                                                                                                                                                                                                                                                                                                                                                                                                                                                                                                                                                                                                                                                                                                                                                                                                                                                                                                                                                                                                                                                                                                                                                                                                                                                                                                                                                                                                                                                                                                                                                                                                                                                                                                                                                                                                                                                                                                                                                                                                                                                                                                                                                                                                                                                                                                                                                                                                                                                                                                                                                                                                                                                                                                                                                                                                                                                                                                                                                                                                                                                                                                                                                                                                                                                                                                                                                                                                                                                                                                                                                                                                                                                                                                                                                                                                                                                                                                                                                                                                                                                                                                                                                                                                                                                                                                                                                                                                                                                                                                                                                                                                                                                                                                                                                                                                                                                                                                                                                                                                                                                                                                                                                                                                                                                                                                                                                                                                                                                                                                                                                                                                                                                                                                                                                                                                                                                                                                                                                                                                                                                                                                                                                                                                                                                                                                                                                                                                                                                                                                                                                                                                                                                                                                                                                                                                                                                                                                                                                                                                                                                                                                                                                                                                                                                                                                                                                                                                                                                                                                                                                                                                                                                                                                                                                                                                                                                                                                                                                                                                                                                                                                                                                                                                                                                                                                                                                                                                                                                                                                                                                                                                                                                                                                                                                                                                                                                                                                                                                                                                                                                                                                                                                                                                                                                                                                                                                                                                                                                                                                                                                                                                                                                                                                                                                                                                                                                                                                                                                                                                                                                                                                                                                                                                                                                                                                                                                                                                                                                                                                                                                                                                                                                                                                                                                                                                                                                                                                                                                                                                                                                                                                                                                                                                                                                                                                                                                                                                                                                                                                                                                                                                                                                                                                                                                                                                                                                                                                                                                                                                                                                                                                                                                                                                                                                                                                                                                                                                                                                                                                                                                                                                                                                                                                                                                                                                                                                                                                                                                                                                                                                                                                                                                                                                                                                                                                                                                                                                                                                                                                                                                                                                                                                                                                                                                                                                                                                                                                                                                                                                                                                                                                                                                                                                                                                                                                                                                                                                                                                                                                                                                                                                                                                                                                                                                                                                                                                                                                                                                                                                                                                                                                                                                                                                                                                                                                                                                                                                                                                                                                                                                                                                                                                                                                                                                                                                                                                                                                                                                                                                                                                                                                                                                                                                                                                                                                                                                                                                                                                                                                                                                                                                                                                                                                                                                                                                                                                                                                                                                                                                                                                                                                                                                                                                                                                                                                                                                                                                                                                                                                                                                                                                                                                                                                                                                                                                                                                                                                                                                                                                                                                                                                                                                                                                                                                                                                                                                                                                                                                                                                                                                                                                                                                                                                                                                                                                                                                                                                                                                                                                                                                                                                                                                                                                                                                                                                                                                                                                                                                                                                                                                                                                                                                                                                                                                                                                                                                                                                                                                                                                                                                                                                                                                                                                                                                                                                                                                                                                                                                                                                                                                                                                                                                                                                                                                                                                                                                                                                                                                                                                                                                                                                                                                                                                                                                                                                                                                                                                                                                                                                                                                                                                                                                                                                                                                                                                                                                                                                                                                                                                                                                                                                                                                                                                                                                                                                                                                                                                                                                                                                                                                                                                                                                                                                                                                                                                                                                                                                                                                                                                                                                                                                                                                                                                                                                                                                                                                                                                                                                                                                                                                                                                                                                                                                                                                                                                                                                                                                                                                                                                                                                                                                                                                                                                                                                                                                                                                                                                                                                                                                                                                                                                                                                                                                                                                                                                                                                                                                                                                                                                                                                                                                                                                                                                                                                                                                                                                                                                                                                                                                                                                                                                                                                                                                                                                                                                                                                                                                                                                                                                                                                                                                                                                                                                                                                                                                                                                                                                                                                                                                                                                                                                                                                                                                                                                                                                                                                                                                                                                                                                                                                                                                                                                                                                                                                                                                                                                                                                                                                                                                                                                                                                                                                                                                                                                                                                                                                                                                                                                                                                                                                                                                                                                                                                                                                                                                                                                                                                                                                                                                                                                                                                                                                                                                                                                                                                                                                                                                                                                                                                                                                                                                                                                                                                                                                                                                                                                                                                                                                                                                                                                                                                                                                                                                                                                                                                                                                                                                                                                                                                                                                                                                                                                                                                                                                                                                                                                                                                                                                                                                                                                                                                                                                                                                                                                                                                                                                                                                                                                                                                                                                                                                                                                                                                                                                                                                                                                                                                                                                                                                                                                                                                                                                                                                                                                                                                                                                                                                                                                                                                                                                                                                                                                                                                                                                                                                                                                                                                                                                                                                                                                                                                                                                                                                                                                                                                                                                                                                                                                                                                                                                                                                                                                                                                                                                                                                                                                                                                                                                                                                                                                                                                                                                                                                                                                                                                                                                                                                                                                                                                                                                                                                                                                                                                                                                                                                                                                                                                                                                                                                                                                                                                                                                                                                                                                                                                                                                                                                                                                                                                                                                                                                                                                                                                                                                                                                                                                                                                                                                                                                                                                                                                                                                                                                                                                                                                                                                                                                                                                                                                                                                                                                                                                                                                                                                                                                                                                                                                                                                                                                                                                                                                                                                                                                                                                                                                                                                                                                                                                                                                                                                                                                                                                                                                                                                                                                                                                                                                                                                                                                                                                                                                                                                                                                                                                                                                                                                                                                                                                                                                                                                                                                                                                                                                                                                                                                                                                                                                                                                                                                                                                                                                                                                                                                                                                                                                                                                                                                                                                                                                                                                                                                                                                                                                                                                                                                                                                                                                                                                                                                                                                                                                                                                                                                                                                                                                                                                                                                                                                                                                                                                                                                                                                                                                                                                                                                                                                                                                                                                                                                                                                                                                                                                                                                                                                                                                                                                                                                                                                                                                                                                                                                                                                                                                                                                                                                                                                                                                                                                                                                                                                                                                                                                                                                                                                                                                                                                                                                                                                                                                                                                                                                                                                                                                                                                                                                                                                                                                                                                                                                                                                                                                                                                                                                                                                                                                                                                                                                                                                                                                                                                                                                                                                                                                                                                                                                                                                                                                                                                                                                                                                                                                                                                                                                                                                                                                                                                                                                                                                                                                                                                                                                                                                                                                                                                                                                                                                                                                                                                                                                                                                                                                                                                                                                                                                                                                                                                                                                                                                                                                                                                                                                                                                                                                                                                                                                                                                                                                                                                                                                                                                                                                                                                                                                                                                                                                                                                                                                                                                                                                                                                                                                                                                                                                                                                                                                                                                                                                                                                                                                                                                                                                                                                                                                                                                                                                                                                                                                                                                                                                                                                                                                                                                                                                                                                                                                                                                                                                                                                                                                                                                                                                                                                                                                                                                                                                                                                                                                                                                                                                                                                                                                                                                                                                                                                                                                                                                                                                                                                                                                                                                                                                                                                                                                                                                                                                                                                                                                                                                                                                                                                                                                                                                                                                                                                                                                                                                                                                                                                                                                                                                                                                                                                                                                                                                                                                                                                                                                                                                                                                                                                                                                                                                                                                                                                                                                                                                                                                                                                                                                                                                                                                                                                                                                                                                                                                               EW := "EW_LF_CM01.BN01",
	                     Messbereich_Min := "Analogwerte"."LF_CM01.BN01".MB_min,
	                     Messbereich_Max := "Analogwerte"."LF_CM01.BN01".MB_max,
	                     UG_Alarm := "Analogwerte"."LF_CM01.BN01".UG_Alarm,
	                     OG_Alarm := "Analogwerte"."LF_CM01.BN01".OG_Alarm,
	                     GF := "Analogwerte"."LF_CM01.BN01".GF,
	                     Al_Drahtbruch => "Analogwerte"."LF_CM01.BN01".Drahtbruch,
	                     Al_MW_ausserhalb => "Analogwerte"."LF_CM01.BN01".ungueltig,
	                     Messwert := "Panel".IW."LF_CM01.BN01");
	        // Leitfähigkeit Düsen Umwälzung
	        "Analogwert"(Deaktiviert:=FALSE,
